PROGRAM Axis04_Z_1
VAR
	Axis04: AXIS_REF;											//회전축
	Axis04_MC_Home: FB_HomeBeforeMoveAX8000:=(channel:=2);
	Axis04_MC_Power: MC_Power;
	Axis04_Status: MC_ReadStatus;
	Axis04_Position_Read: MC_ReadActualPosition;
	Axis04_Velocity_Read: MC_ReadActualVelocity;
	Axis04_Reset: MC_Reset;										//모터 알람 리셋
	Axis04_Stop: MC_Stop;										//모터 정지
	Axis04_Press_Move: MC_MoveAbsolute;
	Axis04_Home_Pos_Move: MC_MoveAbsolute;
	Axis04_Wait_Pos_Move: MC_MoveAbsolute;
	Axis04_Target_Pos_Move: MC_MoveAbsolute;
	Axis04_Work_End_Move: MC_MoveAbsolute;
	Axis04_Jog: MC_Jog;
	
	
	Always_ON	:	BOOL	:=TRUE	;//상시 ON
	Always_OFF	:	BOOL	:=FALSE	;//상시 OFF


	ddd: FB_HomeBeforeMoveAX8000;
	Axis04_Tool_Change: MC_MoveAbsolute;
	TON_555: TON;
	TON_500: TON;
END_VAR
VAR // added by the converter: edge detectors and wires of the graphical bodies
    _rt1, _rt2, _rt3, _rt4, _rt5, _rt6 : R_TRIG;
END_VAR

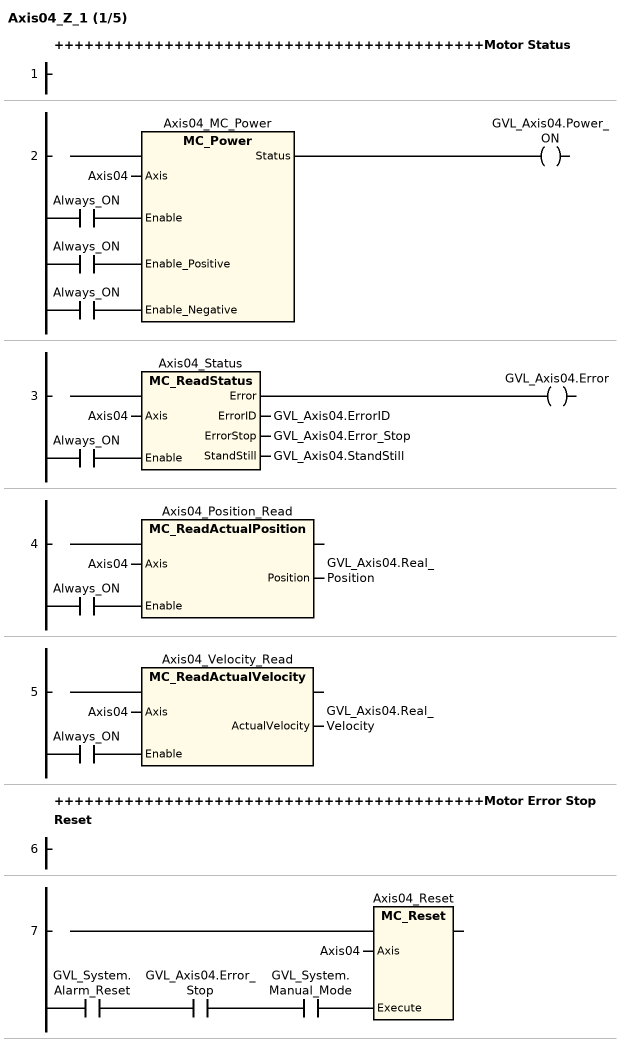
// NETWORK 1: +++++++++++++++++++++++++++++++++++++++++++Motor Status

// NETWORK 2
Axis04_MC_Power(
    Axis := Axis04,
    Enable := Always_ON,
    Enable_Positive := Always_ON,
    Enable_Negative := Always_ON); // MC_Power
GVL_Axis04.Power_ON := Axis04_MC_Power.Status;

// NETWORK 3
Axis04_Status(
    Axis := Axis04,
    Enable := Always_ON,
    Error => GVL_Axis04.Error,
    ErrorID => GVL_Axis04.ErrorID,
    ErrorStop => GVL_Axis04.Error_Stop,
    StandStill => GVL_Axis04.StandStill); // MC_ReadStatus

// NETWORK 4
Axis04_Position_Read(Axis := Axis04, Enable := Always_ON, Position => GVL_Axis04.Real_Position); // MC_ReadActualPosition

// NETWORK 5
Axis04_Velocity_Read(Axis := Axis04, Enable := Always_ON, ActualVelocity => GVL_Axis04.Real_Velocity); // MC_ReadActualVelocity

// NETWORK 6: +++++++++++++++++++++++++++++++++++++++++++Motor Error Stop Reset

// NETWORK 7
Axis04_Reset(Axis := Axis04, Execute := GVL_System.Alarm_Reset AND GVL_Axis04.Error_Stop AND GVL_System.Manual_Mode); // MC_Reset

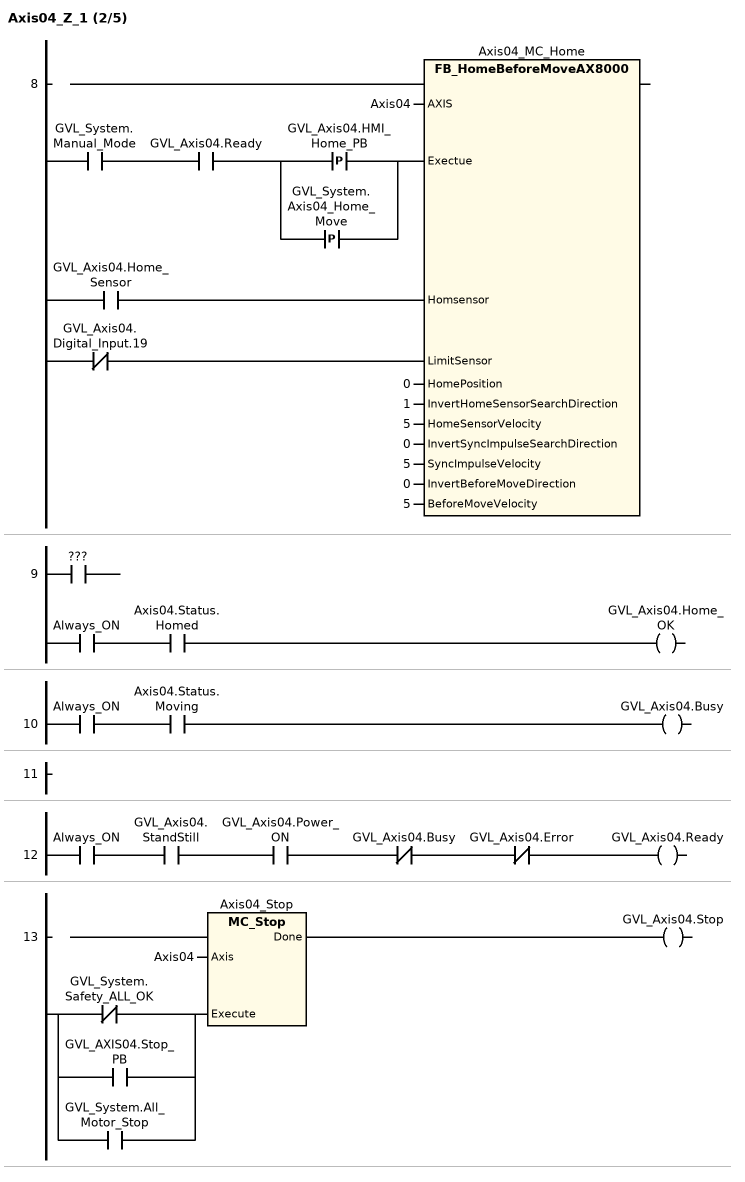
// NETWORK 8
_rt1(CLK := GVL_Axis04.HMI_Home_PB);
_rt2(CLK := GVL_System.Axis04_Home_Move);
Axis04_MC_Home(
    AXIS := Axis04,
    Exectue := GVL_System.Manual_Mode AND GVL_Axis04.Ready AND (_rt1.Q OR _rt2.Q),
    Homsensor := GVL_Axis04.Home_Sensor,
    LimitSensor := NOT GVL_Axis04.Digital_Input.19,
    HomePosition := 0,
    InvertHomeSensorSearchDirection := 1,
    HomeSensorVelocity := 5,
    InvertSyncImpulseSearchDirection := 0,
    SyncImpulseVelocity := 5,
    InvertBeforeMoveDirection := 0,
    BeforeMoveVelocity := 5); // FB_HomeBeforeMoveAX8000

// NETWORK 9
GVL_Axis04.Home_OK := Always_ON AND Axis04.Status.Homed;

// NETWORK 10
GVL_Axis04.Busy := Always_ON AND Axis04.Status.Moving;

// NETWORK 11

// NETWORK 12
GVL_Axis04.Ready := Always_ON AND GVL_Axis04.StandStill AND GVL_Axis04.Power_ON AND NOT GVL_Axis04.Busy AND NOT GVL_Axis04.Error;

// NETWORK 13
Axis04_Stop(Axis := Axis04, Execute := NOT GVL_System.Safety_ALL_OK OR GVL_AXIS04.Stop_PB OR GVL_System.All_Motor_Stop); // MC_Stop
GVL_Axis04.Stop := Axis04_Stop.Done;

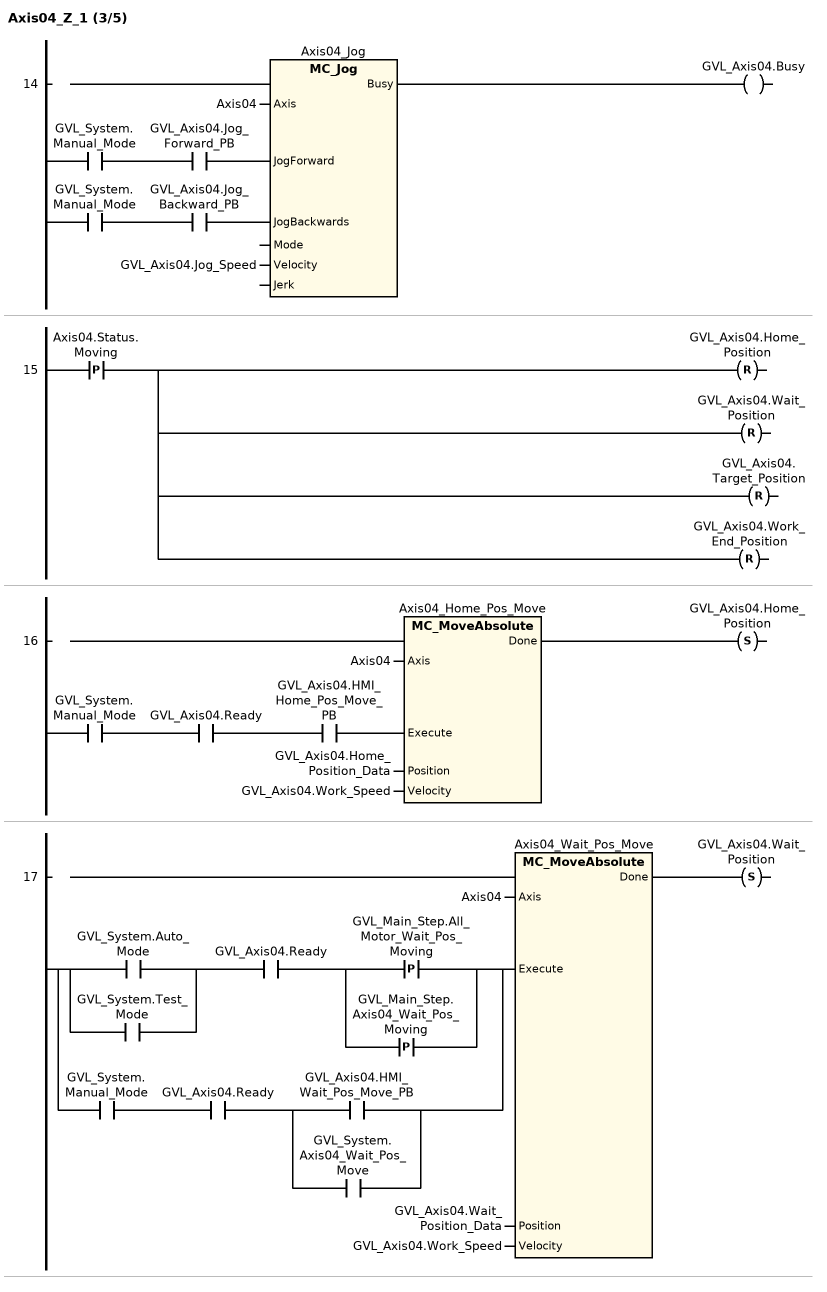
// NETWORK 14
Axis04_Jog(
    Axis := Axis04,
    JogForward := GVL_System.Manual_Mode AND GVL_Axis04.Jog_Forward_PB,
    JogBackwards := GVL_System.Manual_Mode AND GVL_Axis04.Jog_Backward_PB,
    Velocity := GVL_Axis04.Jog_Speed,
    Busy => GVL_Axis04.Busy); // MC_Jog

// NETWORK 15
_rt3(CLK := Axis04.Status.Moving);
GVL_Axis04.Home_Position R= _rt3.Q;
GVL_Axis04.Wait_Position R= _rt3.Q;
GVL_Axis04.Target_Position R= _rt3.Q;
GVL_Axis04.Work_End_Position R= _rt3.Q;

// NETWORK 16
Axis04_Home_Pos_Move(
    Axis := Axis04,
    Execute := GVL_System.Manual_Mode AND GVL_Axis04.Ready AND GVL_Axis04.HMI_Home_Pos_Move_PB,
    Position := GVL_Axis04.Home_Position_Data,
    Velocity := GVL_Axis04.Work_Speed); // MC_MoveAbsolute
GVL_Axis04.Home_Position S= Axis04_Home_Pos_Move.Done;

// NETWORK 17
_rt4(CLK := GVL_Main_Step.All_Motor_Wait_Pos_Moving);
_rt5(CLK := GVL_Main_Step.Axis04_Wait_Pos_Moving);
Axis04_Wait_Pos_Move(
    Axis := Axis04,
    Execute := (GVL_System.Auto_Mode OR GVL_System.Test_Mode) AND GVL_Axis04.Ready AND (_rt4.Q OR _rt5.Q) OR GVL_System.Manual_Mode AND GVL_Axis04.Ready AND (GVL_Axis04.HMI_Wait_Pos_Move_PB OR GVL_System.Axis04_Wait_Pos_Move),
    Position := GVL_Axis04.Wait_Position_Data,
    Velocity := GVL_Axis04.Work_Speed); // MC_MoveAbsolute
GVL_Axis04.Wait_Position S= Axis04_Wait_Pos_Move.Done;

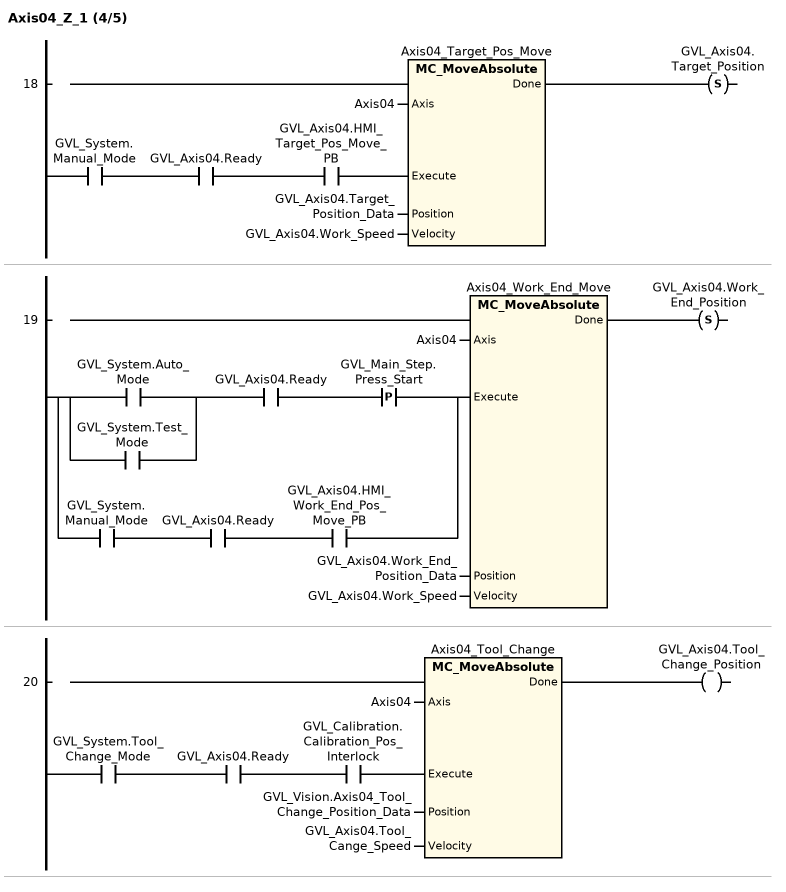
// NETWORK 18
Axis04_Target_Pos_Move(
    Axis := Axis04,
    Execute := GVL_System.Manual_Mode AND GVL_Axis04.Ready AND GVL_Axis04.HMI_Target_Pos_Move_PB,
    Position := GVL_Axis04.Target_Position_Data,
    Velocity := GVL_Axis04.Work_Speed); // MC_MoveAbsolute
GVL_Axis04.Target_Position S= Axis04_Target_Pos_Move.Done;

// NETWORK 19
_rt6(CLK := GVL_Main_Step.Press_Start);
Axis04_Work_End_Move(
    Axis := Axis04,
    Execute := (GVL_System.Auto_Mode OR GVL_System.Test_Mode) AND GVL_Axis04.Ready AND _rt6.Q OR GVL_System.Manual_Mode AND GVL_Axis04.Ready AND GVL_Axis04.HMI_Work_End_Pos_Move_PB,
    Position := GVL_Axis04.Work_End_Position_Data,
    Velocity := GVL_Axis04.Work_Speed); // MC_MoveAbsolute
GVL_Axis04.Work_End_Position S= Axis04_Work_End_Move.Done;

// NETWORK 20
Axis04_Tool_Change(
    Axis := Axis04,
    Execute := GVL_System.Tool_Change_Mode AND GVL_Axis04.Ready AND GVL_Calibration.Calibration_Pos_Interlock,
    Position := GVL_Vision.Axis04_Tool_Change_Position_Data,
    Velocity := GVL_Axis04.Tool_Cange_Speed); // MC_MoveAbsolute
GVL_Axis04.Tool_Change_Position := Axis04_Tool_Change.Done;

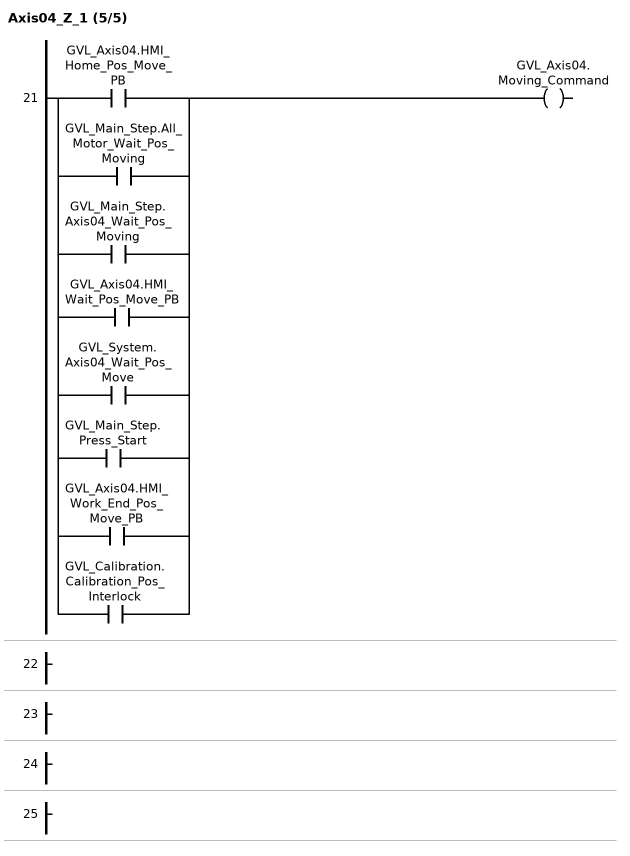
// NETWORK 21
GVL_Axis04.Moving_Command := GVL_Axis04.HMI_Home_Pos_Move_PB OR GVL_Main_Step.All_Motor_Wait_Pos_Moving OR GVL_Main_Step.Axis04_Wait_Pos_Moving OR GVL_Axis04.HMI_Wait_Pos_Move_PB OR GVL_System.Axis04_Wait_Pos_Move OR GVL_Main_Step.Press_Start OR GVL_Axis04.HMI_Work_End_Pos_Move_PB OR GVL_Calibration.Calibration_Pos_Interlock;

// NETWORK 22

// NETWORK 23

// NETWORK 24

// NETWORK 25

END_PROGRAM

(* stored: Version 1.1.0.1, ProductVersion 3.1.4024.15
   POU Axis04_Z_1: Id {2a0472e6-ef59-475e-88bb-8c5956697ac2}, SpecialFunc None *)
